FUNCTION TryConvert_LWORD_TO_STRING : BOOL
VAR_INPUT
	in : LWORD;
	out : REFERENCE TO STRING;
END_VAR

out := LWORD_TO_STRING(in);
TryConvert_LWORD_TO_STRING := TRUE;

END_FUNCTION

(* stored: Version 1.1.0.1, ProductVersion 3.1.4024.12
   POU TryConvert_LWORD_TO_STRING: Id {1634f022-e36f-4266-be18-6ae305f7ee6f}, SpecialFunc None *)
